(* PLC project Generated.project, CODESYS CODESYS V3.5 SP19 Patch 1 *)
(* stored: creationDateTime 2026-07-29T10:44:04.824484, modificationDateTime 2026-07-29T10:44:04.824484 *)

{attribute 'qualified_only'}
{attribute 'strict'}
TYPE E_WinchFinalInterlockState : (DISABLED := 0, READY := 1, WAIT_BRAKE_COMMAND_CONFIRMATION := 2, WAIT_STEP_DELAY := 3, WAIT_RESTART_DELAY := 4, FAULT := 5);
END_TYPE
